// TIA Portal V16 export
// export: Created 2021-12-01T21:19:43.5789487Z, ExportSetting WithDefaults, DisplayName Totally Integrated Automation Portal, DisplayVersion V16 Update 4, DisplayName TIA Portal Version Control Interface, DisplayVersion V16 Update 2, DisplayName TIA Portal Openness, DisplayVersion V16 Update 4, DisplayName SINAMICS Startdrive Advanced, DisplayVersion V16 Update 5, DisplayName SINAMICS Startdrive G130, G150, S120, S150, SINAMICS MV, S210, DisplayVersion V16 Update 5, DisplayName SINAMICS Startdrive G110M, G120, G120C, G120D, G120P, G115D, DisplayVersion V16 Update 5, DisplayName STEP 7 Professional, DisplayVersion V16 Update 4, DisplayName STEP 7 Safety, DisplayVersion V16, DisplayName WinCC Advanced, DisplayVersion V16 Update 4
FUNCTION "ST00242_FC" : Void   // FC62, LAD
TITLE = ST00242
{ S7_Optimized_Access := 'TRUE' }
VERSION : 0.1
// stored: AutoNumber true, IsIECCheckEnabled false, SetENOAutomatically false, UDAEnableTagReadback false
   VAR_IN_OUT
      OPMODE : "OPMODE_OUT_UDT";
      HMI_EXTENSION : "HMI_EXTENSION_PANEL_UDT";
   END_VAR
   VAR_TEMP
      EmptyHS : "RT_HANDSHAKE_UDT";
   END_VAR
BEGIN

REGION Network 1: Alarm
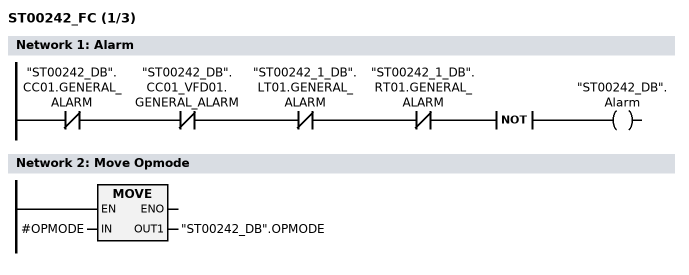
   RUNG wire#powerrail
      I_Contact( "ST00242_DB".CC01.GENERAL_ALARM )
      I_Contact( "ST00242_DB".CC01_VFD01.GENERAL_ALARM )
      I_Contact( "ST00242_1_DB".LT01.GENERAL_ALARM )
      I_Contact( "ST00242_1_DB".RT01.GENERAL_ALARM )
      Not()
      Coil( "ST00242_DB".Alarm )
   END_RUNG
   // the same network as SCL:
   "ST00242_DB".Alarm := NOT (NOT "ST00242_DB".CC01.GENERAL_ALARM AND NOT "ST00242_DB".CC01_VFD01.GENERAL_ALARM AND NOT "ST00242_1_DB".LT01.GENERAL_ALARM AND NOT "ST00242_1_DB".RT01.GENERAL_ALARM);
END_REGION

REGION Network 2: Move Opmode
   RUNG wire#powerrail
      Move(in := #OPMODE, out1 => "ST00242_DB".OPMODE)
   END_RUNG
   // the same network as SCL:
   "ST00242_DB".OPMODE := #OPMODE;
END_REGION

REGION Network 3: *******************CC01 Control*******************
END_REGION

REGION Network 4 (SCL): CC01 Parameters
   //"ST00242_DB".CC01.PARA_SET.Para.StopOnInPos := true;
END_REGION

REGION Network 5: CC01 FB Control
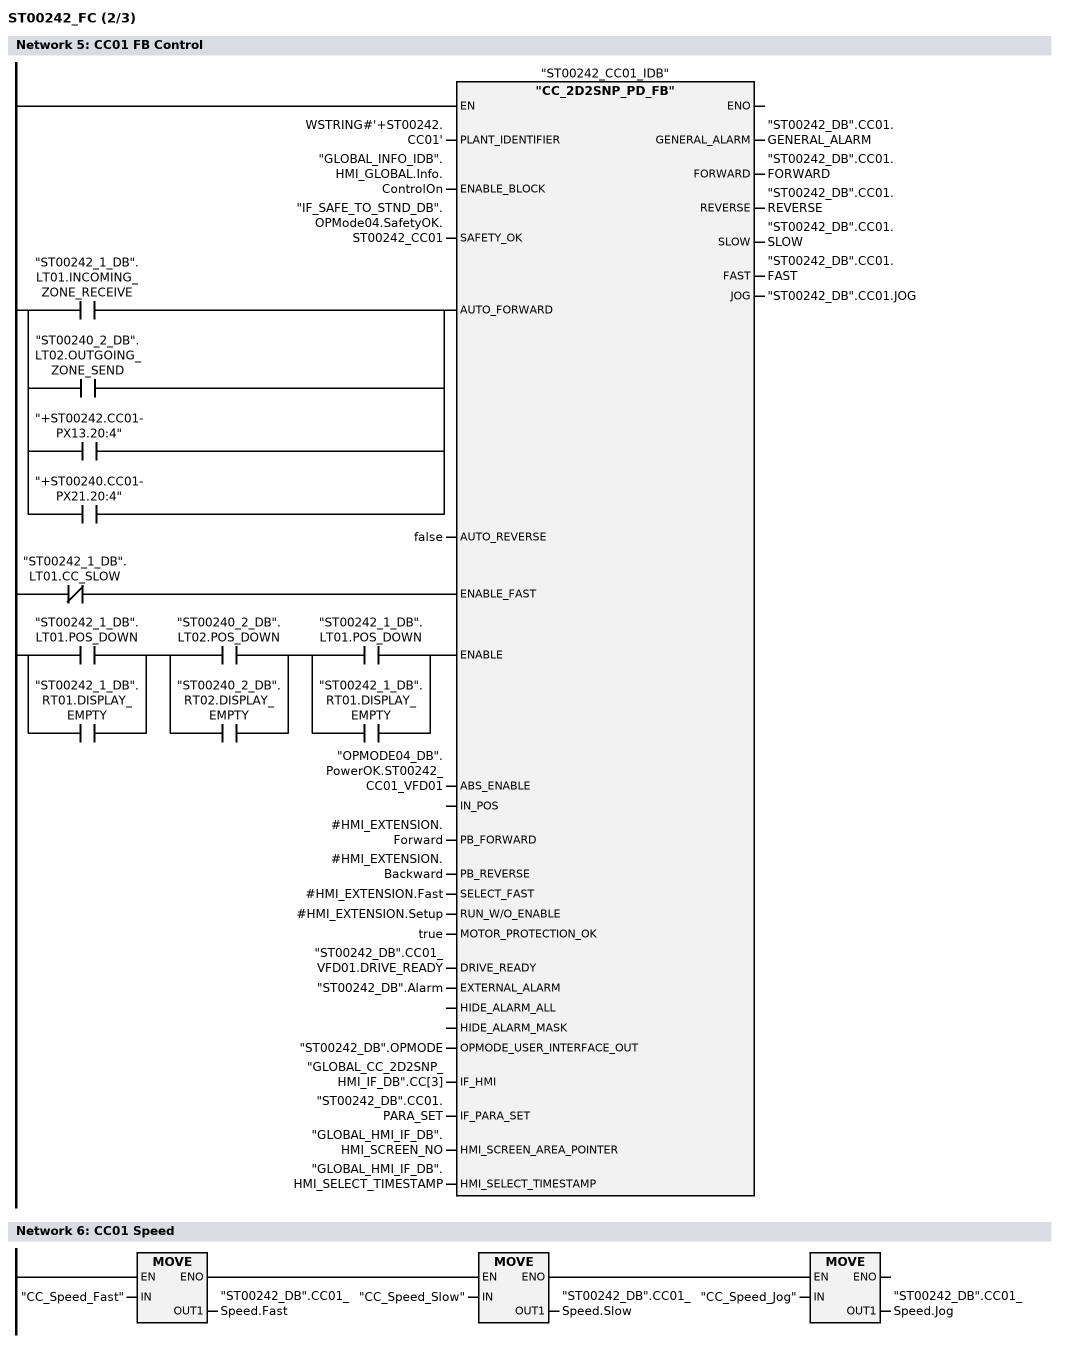
   RUNG wire#powerrail
      "ST00242_CC01_IDB"(AUTO_FORWARD := wire#w1, ENABLE_FAST := wire#w2, ENABLE := wire#w5, PLANT_IDENTIFIER := WSTRING#'+ST00242.CC01', ENABLE_BLOCK := "GLOBAL_INFO_IDB".HMI_GLOBAL.Info.ControlOn, SAFETY_OK := "IF_SAFE_TO_STND_DB".OPMode04.SafetyOK.ST00242_CC01, AUTO_REVERSE := false, ABS_ENABLE := "OPMODE04_DB".PowerOK.ST00242_CC01_VFD01, IN_POS :=, PB_FORWARD := #HMI_EXTENSION.Forward, PB_REVERSE := #HMI_EXTENSION.Backward, SELECT_FAST := #HMI_EXTENSION.Fast, "RUN_W/O_ENABLE" := #HMI_EXTENSION.Setup, MOTOR_PROTECTION_OK := true, DRIVE_READY := "ST00242_DB".CC01_VFD01.DRIVE_READY, EXTERNAL_ALARM := "ST00242_DB".Alarm, HIDE_ALARM_ALL :=, HIDE_ALARM_MASK :=, OPMODE_USER_INTERFACE_OUT := "ST00242_DB".OPMODE, IF_HMI := "GLOBAL_CC_2D2SNP_HMI_IF_DB".CC[3], IF_PARA_SET := "ST00242_DB".CC01.PARA_SET, HMI_SCREEN_AREA_POINTER := "GLOBAL_HMI_IF_DB".HMI_SCREEN_NO, HMI_SELECT_TIMESTAMP := "GLOBAL_HMI_IF_DB".HMI_SELECT_TIMESTAMP, GENERAL_ALARM => "ST00242_DB".CC01.GENERAL_ALARM, FORWARD => "ST00242_DB".CC01.FORWARD, REVERSE => "ST00242_DB".CC01.REVERSE, SLOW => "ST00242_DB".CC01.SLOW, FAST => "ST00242_DB".CC01.FAST, JOG => "ST00242_DB".CC01.JOG)
   END_RUNG
   RUNG wire#powerrail
      Contact( "ST00242_1_DB".LT01.INCOMING_ZONE_RECEIVE )
   END_RUNG wire#w1
   RUNG wire#powerrail
      Contact( "ST00240_2_DB".LT02.OUTGOING_ZONE_SEND )
   END_RUNG wire#w1
   RUNG wire#powerrail
      Contact( "+ST00242.CC01-PX13.20:4" )
   END_RUNG wire#w1
   RUNG wire#powerrail
      Contact( "+ST00240.CC01-PX21.20:4" )
   END_RUNG wire#w1
   RUNG wire#powerrail
      I_Contact( "ST00242_1_DB".LT01.CC_SLOW )
   END_RUNG wire#w2
   RUNG wire#powerrail
      Contact( "ST00242_1_DB".LT01.POS_DOWN )
      wire#w3
      Contact( "ST00240_2_DB".LT02.POS_DOWN )
      wire#w4
      Contact( "ST00242_1_DB".LT01.POS_DOWN )
   END_RUNG wire#w5
   RUNG wire#powerrail
      Contact( "ST00242_1_DB".RT01.DISPLAY_EMPTY )
   END_RUNG wire#w3
   RUNG wire#w3
      Contact( "ST00240_2_DB".RT02.DISPLAY_EMPTY )
   END_RUNG wire#w4
   RUNG wire#w4
      Contact( "ST00242_1_DB".RT01.DISPLAY_EMPTY )
   END_RUNG wire#w5
   // the same network as SCL:
   "ST00242_CC01_IDB"(PLANT_IDENTIFIER := WSTRING#'+ST00242.CC01',   // "CC_2D2SNP_PD_FB"
                      ENABLE_BLOCK := "GLOBAL_INFO_IDB".HMI_GLOBAL.Info.ControlOn,
                      SAFETY_OK := "IF_SAFE_TO_STND_DB".OPMode04.SafetyOK.ST00242_CC01,
                      AUTO_FORWARD := "ST00242_1_DB".LT01.INCOMING_ZONE_RECEIVE OR "ST00240_2_DB".LT02.OUTGOING_ZONE_SEND OR "+ST00242.CC01-PX13.20:4" OR "+ST00240.CC01-PX21.20:4",
                      AUTO_REVERSE := false,
                      ENABLE_FAST := NOT "ST00242_1_DB".LT01.CC_SLOW,
                      ENABLE := ("ST00242_1_DB".LT01.POS_DOWN OR "ST00242_1_DB".RT01.DISPLAY_EMPTY) AND ("ST00240_2_DB".LT02.POS_DOWN OR "ST00240_2_DB".RT02.DISPLAY_EMPTY) AND ("ST00242_1_DB".LT01.POS_DOWN OR "ST00242_1_DB".RT01.DISPLAY_EMPTY),
                      ABS_ENABLE := "OPMODE04_DB".PowerOK.ST00242_CC01_VFD01,
                      PB_FORWARD := #HMI_EXTENSION.Forward,
                      PB_REVERSE := #HMI_EXTENSION.Backward,
                      SELECT_FAST := #HMI_EXTENSION.Fast,
                      "RUN_W/O_ENABLE" := #HMI_EXTENSION.Setup,
                      MOTOR_PROTECTION_OK := true,
                      DRIVE_READY := "ST00242_DB".CC01_VFD01.DRIVE_READY,
                      EXTERNAL_ALARM := "ST00242_DB".Alarm,
                      OPMODE_USER_INTERFACE_OUT := "ST00242_DB".OPMODE,
                      IF_HMI := "GLOBAL_CC_2D2SNP_HMI_IF_DB".CC[3],
                      IF_PARA_SET := "ST00242_DB".CC01.PARA_SET,
                      HMI_SCREEN_AREA_POINTER := "GLOBAL_HMI_IF_DB".HMI_SCREEN_NO,
                      HMI_SELECT_TIMESTAMP := "GLOBAL_HMI_IF_DB".HMI_SELECT_TIMESTAMP,
                      GENERAL_ALARM => "ST00242_DB".CC01.GENERAL_ALARM,
                      FORWARD => "ST00242_DB".CC01.FORWARD,
                      REVERSE => "ST00242_DB".CC01.REVERSE,
                      SLOW => "ST00242_DB".CC01.SLOW,
                      FAST => "ST00242_DB".CC01.FAST,
                      JOG => "ST00242_DB".CC01.JOG);
END_REGION

REGION Network 6: CC01 Speed
   RUNG wire#powerrail
      Move(in := "CC_Speed_Fast", out1 => "ST00242_DB".CC01_Speed.Fast)
      Move(in := "CC_Speed_Slow", out1 => "ST00242_DB".CC01_Speed.Slow)
      Move(in := "CC_Speed_Jog", out1 => "ST00242_DB".CC01_Speed.Jog)
   END_RUNG
   // the same network as SCL:
   "ST00242_DB".CC01_Speed.Fast := "CC_Speed_Fast";
   "ST00242_DB".CC01_Speed.Slow := "CC_Speed_Slow";
   "ST00242_DB".CC01_Speed.Jog := "CC_Speed_Jog";
END_REGION

REGION Network 7: CC01 Drive
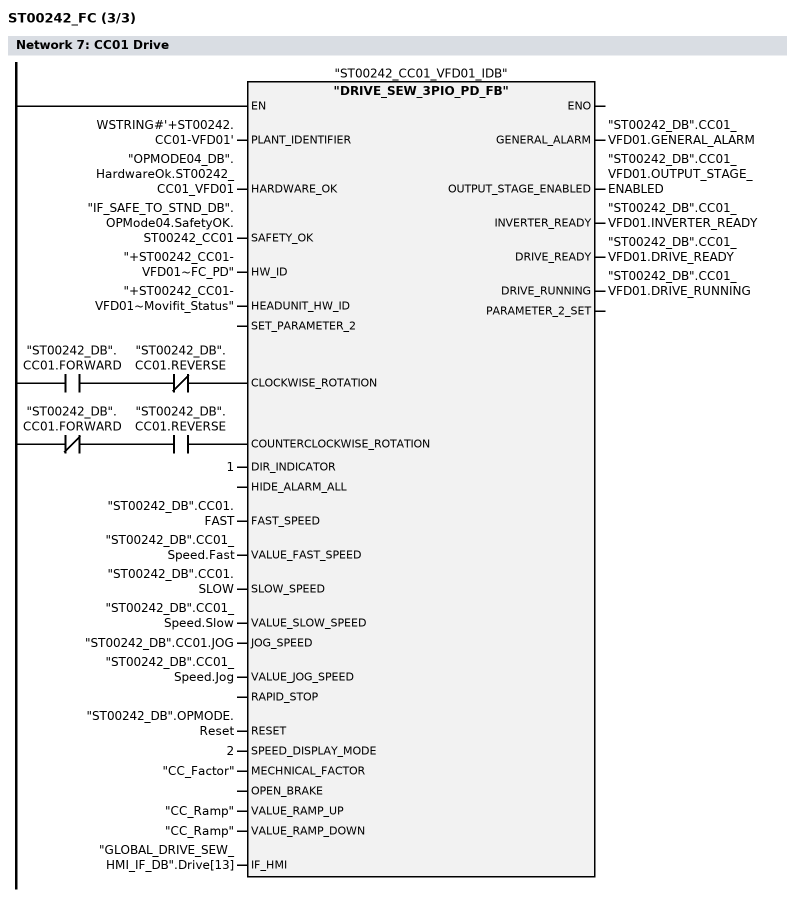
   RUNG wire#powerrail
      "ST00242_CC01_VFD01_IDB"(CLOCKWISE_ROTATION := wire#w1, COUNTERCLOCKWISE_ROTATION := wire#w2, PLANT_IDENTIFIER := WSTRING#'+ST00242.CC01-VFD01', HARDWARE_OK := "OPMODE04_DB".HardwareOk.ST00242_CC01_VFD01, SAFETY_OK := "IF_SAFE_TO_STND_DB".OPMode04.SafetyOK.ST00242_CC01, HW_ID := "+ST00242_CC01-VFD01~FC_PD", HEADUNIT_HW_ID := "+ST00242_CC01-VFD01~Movifit_Status", SET_PARAMETER_2 :=, DIR_INDICATOR := 1, HIDE_ALARM_ALL :=, FAST_SPEED := "ST00242_DB".CC01.FAST, VALUE_FAST_SPEED := "ST00242_DB".CC01_Speed.Fast, SLOW_SPEED := "ST00242_DB".CC01.SLOW, VALUE_SLOW_SPEED := "ST00242_DB".CC01_Speed.Slow, JOG_SPEED := "ST00242_DB".CC01.JOG, VALUE_JOG_SPEED := "ST00242_DB".CC01_Speed.Jog, RAPID_STOP :=, RESET := "ST00242_DB".OPMODE.Reset, SPEED_DISPLAY_MODE := 2, MECHNICAL_FACTOR := "CC_Factor", OPEN_BRAKE :=, VALUE_RAMP_UP := "CC_Ramp", VALUE_RAMP_DOWN := "CC_Ramp", IF_HMI := "GLOBAL_DRIVE_SEW_HMI_IF_DB".Drive[13], GENERAL_ALARM => "ST00242_DB".CC01_VFD01.GENERAL_ALARM, OUTPUT_STAGE_ENABLED => "ST00242_DB".CC01_VFD01.OUTPUT_STAGE_ENABLED, INVERTER_READY => "ST00242_DB".CC01_VFD01.INVERTER_READY, DRIVE_READY => "ST00242_DB".CC01_VFD01.DRIVE_READY, DRIVE_RUNNING => "ST00242_DB".CC01_VFD01.DRIVE_RUNNING, PARAMETER_2_SET =>)
   END_RUNG
   RUNG wire#powerrail
      Contact( "ST00242_DB".CC01.FORWARD )
      I_Contact( "ST00242_DB".CC01.REVERSE )
   END_RUNG wire#w1
   RUNG wire#powerrail
      I_Contact( "ST00242_DB".CC01.FORWARD )
      Contact( "ST00242_DB".CC01.REVERSE )
   END_RUNG wire#w2
   // the same network as SCL:
   "ST00242_CC01_VFD01_IDB"(PLANT_IDENTIFIER := WSTRING#'+ST00242.CC01-VFD01',   // "DRIVE_SEW_3PIO_PD_FB"
                           HARDWARE_OK := "OPMODE04_DB".HardwareOk.ST00242_CC01_VFD01,
                           SAFETY_OK := "IF_SAFE_TO_STND_DB".OPMode04.SafetyOK.ST00242_CC01,
                           HW_ID := "+ST00242_CC01-VFD01~FC_PD",
                           HEADUNIT_HW_ID := "+ST00242_CC01-VFD01~Movifit_Status",
                           CLOCKWISE_ROTATION := "ST00242_DB".CC01.FORWARD AND NOT "ST00242_DB".CC01.REVERSE,
                           COUNTERCLOCKWISE_ROTATION := NOT "ST00242_DB".CC01.FORWARD AND "ST00242_DB".CC01.REVERSE,
                           DIR_INDICATOR := 1,
                           FAST_SPEED := "ST00242_DB".CC01.FAST,
                           VALUE_FAST_SPEED := "ST00242_DB".CC01_Speed.Fast,
                           SLOW_SPEED := "ST00242_DB".CC01.SLOW,
                           VALUE_SLOW_SPEED := "ST00242_DB".CC01_Speed.Slow,
                           JOG_SPEED := "ST00242_DB".CC01.JOG,
                           VALUE_JOG_SPEED := "ST00242_DB".CC01_Speed.Jog,
                           RESET := "ST00242_DB".OPMODE.Reset,
                           SPEED_DISPLAY_MODE := 2,
                           MECHNICAL_FACTOR := "CC_Factor",
                           VALUE_RAMP_UP := "CC_Ramp",
                           VALUE_RAMP_DOWN := "CC_Ramp",
                           IF_HMI := "GLOBAL_DRIVE_SEW_HMI_IF_DB".Drive[13],
                           GENERAL_ALARM => "ST00242_DB".CC01_VFD01.GENERAL_ALARM,
                           OUTPUT_STAGE_ENABLED => "ST00242_DB".CC01_VFD01.OUTPUT_STAGE_ENABLED,
                           INVERTER_READY => "ST00242_DB".CC01_VFD01.INVERTER_READY,
                           DRIVE_READY => "ST00242_DB".CC01_VFD01.DRIVE_READY,
                           DRIVE_RUNNING => "ST00242_DB".CC01_VFD01.DRIVE_RUNNING);
END_REGION
END_FUNCTION
